Yaskawa INFORM job: FMTV_HOOD_FRONT.JBI

/JOB
//NAME FMTV_HOOD_FRONT
//POS
///NPOS 42,0,0,0,0,0
///TOOL 0
///POSTYPE PULSE
///PULSE
C00000=-147066,-165395,-6439,251998,122776,-36821
C00001=-162933,-163816,-54723,90026,118426,-23586
C00002=62081,-155211,-116273,69555,-58084,-78743
C00003=85760,-87684,-81866,-22659,-21113,-109718
C00004=72882,-73373,-60477,-37107,-28604,-101540
C00005=71023,-70818,-56661,-38480,-29879,-100787
C00006=18574,-104993,-65177,-61110,-65980,-90833
C00007=18910,-106941,-63431,-53343,-65090,-93083
C00008=19949,-109437,-60928,-41556,-64483,-96452
C00009=21046,-111457,-59722,-32869,-64585,-98875
C00010=21653,-113260,-58584,-24966,-65360,-100914
C00011=14332,-114467,-56294,-20276,-69094,-99993
C00012=7125,-115250,-54652,-16387,-71539,-98606
C00013=7122,-115222,-54628,-16389,-71538,-98604
C00014=4104,-115434,-54308,-18070,-72329,-97644
C00015=1660,-115522,-53193,-19373,-73370,-96958
C00016=1661,-115545,-53213,-19372,-73372,-96959
C00017=1659,-115475,-53152,-19374,-73367,-96957
C00018=1641,-115458,-53123,-19383,-73375,-96953
C00019=-2509,-115720,-52266,-21599,-74766,-95738
C00020=-2479,-118913,-55165,-21562,-74933,-95786
C00021=18019,-118978,-54156,5064,-74006,-104965
C00022=16807,-114856,-50350,4381,-73738,-104569
C00023=-37500,-112729,-50726,-25449,-78492,-86525
C00024=-39204,-115969,-53898,-26278,-79004,-86029
C00025=-23533,-118644,-54295,-5901,-73743,-92892
C00026=-22218,-114834,-50761,-5157,-73480,-93327
C00027=-24545,-114809,-51154,-6487,-73415,-92529
C00028=-26294,-114418,-51842,-7502,-72994,-91898
C00029=-26295,-114418,-51842,-7502,-72995,-91898
C00030=-26254,-114310,-51744,-7478,-72986,-91912
C00031=-27866,-114084,-52870,-8429,-72445,-91305
C00032=-30126,-113522,-53229,-9730,-72193,-90484
C00033=-54961,-106888,-53939,-23561,-72970,-81404
C00034=-70548,-89870,-47676,-31853,-72658,-66323
C00035=-73909,-92553,-51946,-33448,-73201,-65010
C00036=-40956,-108858,-62331,15535,-58796,-95874
C00037=-38939,-103194,-56445,16883,-59198,-96671
C00038=-80173,-70158,-49239,-14673,-45057,-77320
C00039=-81466,-65601,-49747,-10471,-38304,-78559
C00040=-83000,-68132,-53893,-12181,-37749,-77477
C00041=-99132,-82437,-80579,-37363,-43577,-63256
//INST
///DATE 2023/03/28 15:22
///ATTR SC,RW
///GROUP1 RB1
NOP
MOVJ C00000 VJ=65.00  //FROM LEFT
MOVJ C00001 VJ=65.00
MOVJ C00002 VJ=65.00
MOVJ C00003 VJ=65.00  //ABOVE
MOVL C00004 V=65.0  //UP TO
MOVL C00005 V=15.0  //INTO
MOVL C00006 V=15.0
MOVL C00007 V=15.0
MOVL C00008 V=15.0
MOVL C00009 V=15.0
MOVL C00010 V=15.0
MOVL C00011 V=15.0
MOVL C00012 V=15.0
MOVC C00013 V=15.0
MOVC C00014 V=15.0
MOVC C00015 V=15.0
MOVL C00016 V=15.0
MOVC C00017 V=15.0
MOVC C00018 V=15.0
MOVC C00019 V=15.0
MOVL C00020 V=45.0
MOVL C00021 V=45.0
MOVL C00022 V=15.0
MOVL C00023 V=15.0
MOVL C00024 V=45.0
MOVL C00025 V=45.0
MOVC C00026 V=15.0
MOVC C00027 V=15.0
MOVC C00028 V=15.0
MOVL C00029 V=15.0
MOVC C00030 V=15.0
MOVC C00031 V=15.0
MOVC C00032 V=15.0
MOVL C00033 V=15.0  //TO ANGLE
MOVL C00034 V=15.0  //END ANGLE
MOVL C00035 V=15.0  //OUT
MOVL C00036 V=65.0
MOVL C00037 V=15.0
MOVL C00038 V=15.0
MOVL C00039 V=15.0  //END
MOVL C00040 V=15.0  //OUT
MOVL C00041 V=65.0  //AWAY
END
